// TIA Portal V20 export
TYPE "UDT_Accesos"
   STRUCT
      Memorias : Struct
         MPeticion : Bool;
         MPermiso : Bool;
         MEntradaPeticion : Bool;
         Libre_03 : Bool;
         Libre_04 : Bool;
         Libre_05 : Bool;
         TodasMesas_EnParo : Bool;
         AlgunaMesa_EnMarcha : Bool;
         MFP_ParoBlando : Bool;
         MFP_Marcha : Bool;
         MFP_PulsadorPeticion : Bool;
         Libre_13 : Bool;
         Libre_14 : Bool;
         Libre_15 : Bool;
         Libre_16 : Bool;
         Libre_17 : Bool;
      END_STRUCT;
      Mesas : Array[1..20] of UInt;
   END_STRUCT;
END_TYPE
